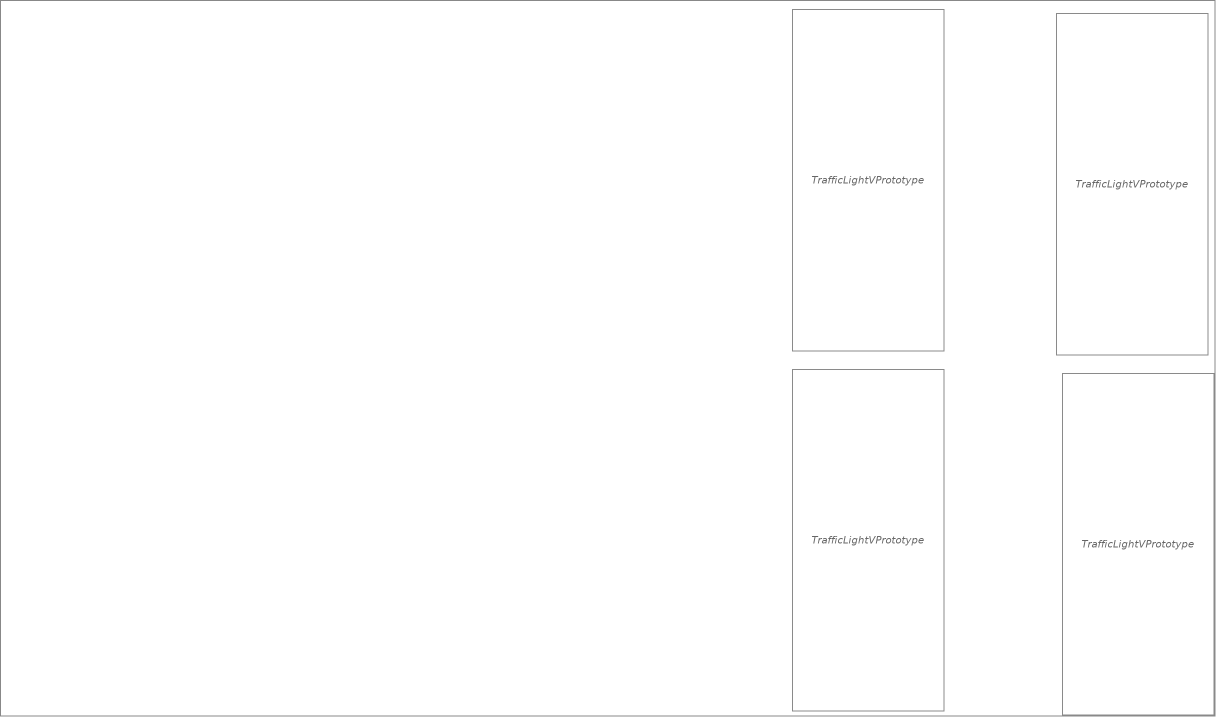
VISUALIZATION TrafficLightV1  // 1216x717
    Frame (792,369 152x342)
        shows TrafficLightVPrototype(stTrafficOut := MAIN.fbCrossing1.fbTrafficLightArray[1].stTrafficLightOutput)
    Frame (1062,373 152x342)
        shows TrafficLightVPrototype(stTrafficOut := MAIN.fbCrossing1.fbTrafficLightArray[3].stTrafficLightOutput)
    Frame (792,9 152x342)
        shows TrafficLightVPrototype(stTrafficOut := MAIN.fbCrossing1.fbTrafficLightArray[4].stTrafficLightOutput)
    Frame (1056,13 152x342)
        shows TrafficLightVPrototype(stTrafficOut := MAIN.fbCrossing1.fbTrafficLightArray[2].stTrafficLightOutput)
END_VISUALIZATION

(* stored: Version 1.1.0.1, ProductVersion 3.1.4024.0
   Visu TrafficLightV1: Id {776f7eae-3eff-4e66-8da1-b388e5f0177d} *)
